// TIA Portal V17 export
// export: Created 2024-08-26T21:07:17.6856096Z, ExportSetting WithDefaults, DisplayName Totally Integrated Automation Portal, DisplayVersion V17 Update 7, DisplayName TIA Portal Openness, DisplayVersion V17 Update 7, DisplayName TIA Portal Version Control Interface, DisplayVersion V17, DisplayName SINAMICS Startdrive Advanced, DisplayVersion V17 SP2, DisplayName SINAMICS Startdrive G110M, G120, G120C, G120D, G120P, G115D, DisplayVersion V17 SP2, DisplayName SINAMICS Startdrive G130, G150, S120, S150, SINAMICS MV, S210, DisplayVersion V17 SP2, DisplayName STEP 7 Professional, DisplayVersion V17 Update 7, DisplayName STEP 7 Safety, DisplayVersion V17 Update 6, DisplayName WinCC Advanced / Unified PC, DisplayVersion V17 Update 7
DATA_BLOCK "Conveyor_DB"   // DB41
{ S7_Optimized_Access := 'FALSE' }
VERSION : 0.1
// stored: AutoNumber true, DBAccessibleFromOPCUA true, DBAccessibleFromWebserver true, IsOnlyStoredInLoadMemory false, IsWriteProtectedInAS false
   VAR
      printLabel : Bool := FALSE;
      description : String := 'BACKREST W33A POWER MEMO L6';
      partNumber : String := '2389161X-01';
      lastScann : String := '038040781M41839';
      okModelBit : Bool := FALSE;
      leftTrackScan : String := 'JI2U07619706';
      rightTrackScan : String := 'FR2I01420707';
      motorScan : String := '038040781M41839';
   END_VAR
BEGIN
END_DATA_BLOCK
